// LS Electric XG5000 project: 레이싱
// PLC LSPLC
// module base 0 slot 0: 입출력 모듈:XBC-DR14E (DC 24V 입력 8점, 릴레이 출력 6점)

PROGRAM NewProgram (task: 스캔 프로그램)

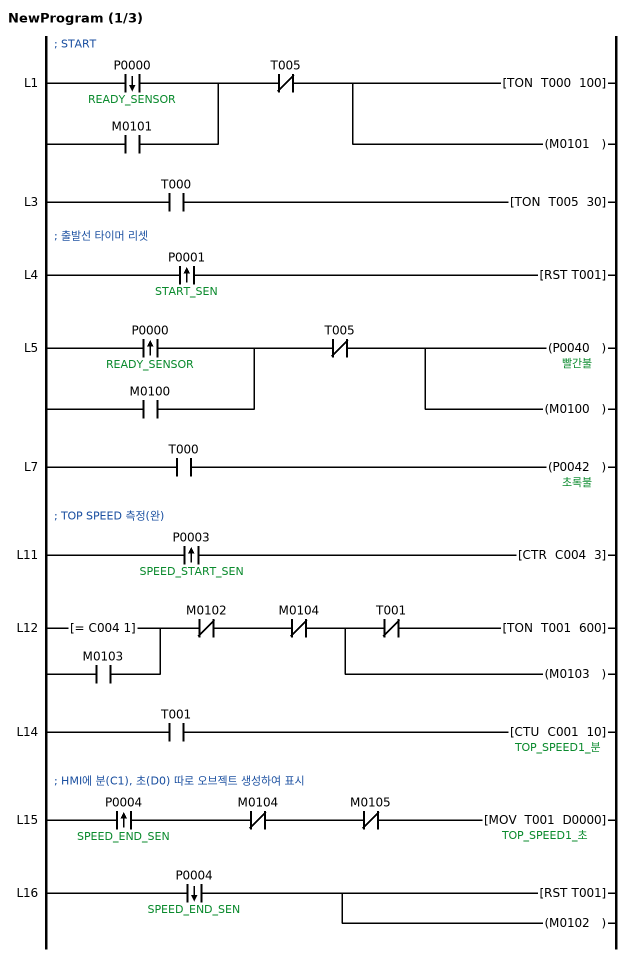
// START
; L1
LOADN     P0000	// READY_SENSOR
OR        M0101
AND NOT   T005
TON       T000 100
OUT       M0101
; L3
LOAD      T000
TON       T005 30
; L4
LOADP     P0001	// START_SEN
RST       T001
// output comment: 출발선 타이머 리셋
; L5
LOADP     P0000	// READY_SENSOR
OR        M0100
AND NOT   T005
OUT       P0040	// 빨간불
OUT       M0100
; L7
LOAD      T000
OUT       P0042	// 초록불
// TOP SPEED 측정(완)
; L11
LOADP     P0003	// SPEED_START_SEN
CTR       C004 3
; L12
LOAD=     C004 1
OR        M0103
AND NOT   M0102
AND NOT   M0104
MPUSH
AND NOT   T001
TON       T001 600
MPOP
OUT       M0103
; L14
LOAD      T001
CTU       C001 10	// TOP_SPEED1_분
; L15
LOADP     P0004	// SPEED_END_SEN
AND NOT   M0104
AND NOT   M0105
MOV       T001 D0000	// TOP_SPEED1_초
// output comment: HMI에 분(C1), 초(D0) 따로 오브젝트 생성하여 표시
; L16
LOADN     P0004	// SPEED_END_SEN
RST       T001
OUT       M0102

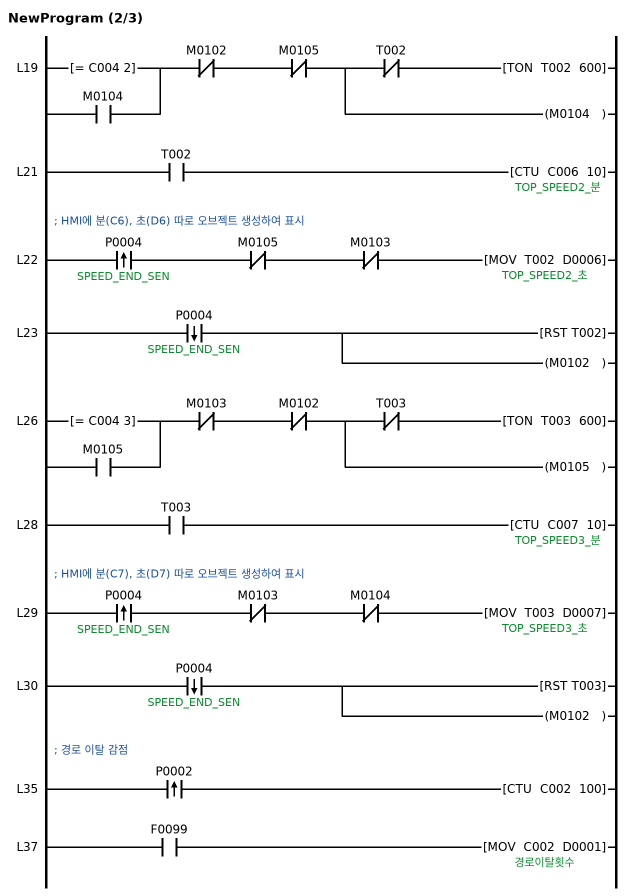
; L19
LOAD=     C004 2
OR        M0104
AND NOT   M0102
AND NOT   M0105
MPUSH
AND NOT   T002
TON       T002 600
MPOP
OUT       M0104
; L21
LOAD      T002
CTU       C006 10	// TOP_SPEED2_분
; L22
LOADP     P0004	// SPEED_END_SEN
AND NOT   M0105
AND NOT   M0103
MOV       T002 D0006	// TOP_SPEED2_초
// output comment: HMI에 분(C6), 초(D6) 따로 오브젝트 생성하여 표시
; L23
LOADN     P0004	// SPEED_END_SEN
RST       T002
OUT       M0102
; L26
LOAD=     C004 3
OR        M0105
AND NOT   M0103
AND NOT   M0102
MPUSH
AND NOT   T003
TON       T003 600
MPOP
OUT       M0105
; L28
LOAD      T003
CTU       C007 10	// TOP_SPEED3_분
; L29
LOADP     P0004	// SPEED_END_SEN
AND NOT   M0103
AND NOT   M0104
MOV       T003 D0007	// TOP_SPEED3_초
// output comment: HMI에 분(C7), 초(D7) 따로 오브젝트 생성하여 표시
; L30
LOADN     P0004	// SPEED_END_SEN
RST       T003
OUT       M0102
// 경로 이탈 감점
; L35
LOADP     P0002
CTU       C002 100
; L37
LOAD      F0099
MOV       C002 D0001	// 경로이탈횟수

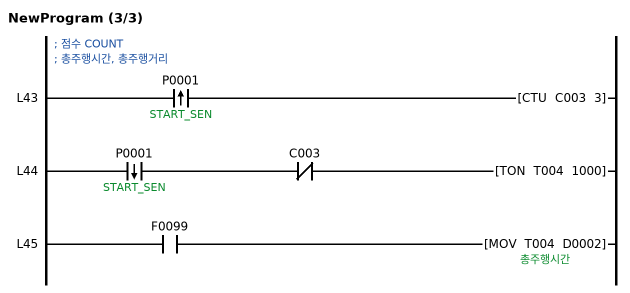
// 점수 COUNT
// 총주행시간, 총주행거리
; L43
LOADP     P0001	// START_SEN
CTU       C003 3
; L44
LOADN     P0001	// START_SEN
AND NOT   C003
TON       T004 1000
; L45
LOAD      F0099
MOV       T004 D0002	// 총주행시간

VARIABLES AND COMMENTS (devices not used above)
P00041	BIT	주황불
C0000	BIT/WORD	출발감점